# EPICS substitutions: SYMETRIE_EPICSApp/Db/SymetriePmac.substitutions
file "$(MOTOR)/db/SymetriePmac.template"
{
pattern
{}
{}
}

file "$(MOTOR)/db/SymetriePmacAxis.template"
{
pattern
{AXIS}
{0}
{1}
{2}
{3}
{4}
{5}
}

file "$(MOTOR)/db/SymetriePmacError.template"
{
pattern
{ADDR}
{0}
{1}
{2}
{3}
{4}
{5}
{6}
{7}
{8}
{9}
{10}
{11}
{12}
{13}
{14}
{15}
{16}
{17}
{18}
{19}
}
